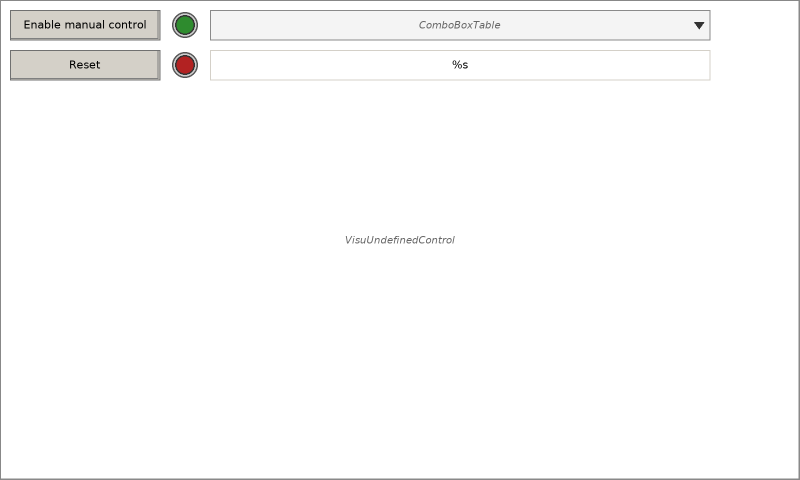
VISUALIZATION ManualControl  // 800x480
VAR_IN_OUT
	stHMI : UDT_HMI_ManualControl;
	fbManualController : FB_ManualController; // Only needed to reference the device array and its size
END_VAR
    Frame (0,0 800x480), input disabled if: NOT stHMI.bEnabled, frame switch variable: stHMI.refSelectedDevice.eDevType
        shows VisuUndefinedControl()
        shows VisuValveControl(pDev := stHMI.pDevValve)
        shows VisuCylinderControl(pDev := stHMI.pDevCylinder)
        shows VisuAxisControl(pDev := stHMI.pDevAxis)
        shows VisuPushbuttonLightControl(pDev := stHMI.pDevPBL)
        shows VisuDigitalInputControl(pDev := stHMI.pDevDigitalInput)
        shows VisuAnlogInputControl(pDev := stHMI.pDevAnalogInput)
        shows VisuDigitalOutControl(pDev := stHMI.pDevDigitalOut)
        shows VisuAnalogOutControl(pDev := stHMI.pDevAnalogOut)
        shows VisuPWMControl(pDev := stHMI.pDevPWMController)
        shows VisuDoublePWMControl(pDev := stHMI.pDevDoublePWM)
        shows VisuEncoderInput(pDev := stHMI.pDevEncoder)
        shows VisuAnalogAxisControl(pDev := stHMI.pDevAnalogAxis)
        shows VisuTwoVelocityAxisControl(pDev := stHMI.pDevTwoVelocityAxis)
        shows VisuKL5151Control(pDev := stHMI.pDevKL5151)
        shows VisuKL15XXControl(pDev := stHMI.pDevKL1512)
        pReferences[2]: HMI=stHMI
        pReferences[3]: HMI=stHMI
        pReferences[4]: HMI=stHMI
        pReferences[5]: HMI=stHMI
        pReferences[6]: HMI=stHMI
        pReferences[7]: HMI=stHMI
        pReferences[8]: HMI=stHMI
        pReferences[9]: HMI=stHMI
        pReferences[10]: HMI=stHMI
        pReferences[11]: HMI=stHMI
        pReferences[12]: HMI=stHMI
        pReferences[13]: HMI=stHMI
        pReferences[14]: HMI=stHMI
        pReferences[15]: HMI=stHMI
    Lamp1 (170,50 30x30), tooltip "component fault active", variable: stHMI.refSelectedDevice.bErrorActive, style: Lamp-Lamp1-Red
    Lamp1 (170,10 30x30), tooltip "Manual control active", variable: stHMI.bEnabled, style: Lamp-Lamp1-Green
    Textfield (210,50 500x30), "%s", text variable: stHMI.refSelectedDevice.sActiveState
    Button (10,50 150x30), "Reset"
        tap stHMI.bReset
    ComboBoxTable (210,10 500x30), variable: stHMI.nSelectedDevice, data array: fbManualController.arDeviceArray
        p1128707560: fbManualController.nNumberOfDevices
        p3854506369: fbManualController.arDeviceArray[INDEX].sName
        p1892666644: fbManualController.arDeviceArray[INDEX].sType
        p338671338: fbManualController.arDeviceArray[INDEX].pFunction^
    Button (10,10 150x30), "Enable manual control"
        toggle stHMI.bEnabled
END_VISUALIZATION

(* stored: Version 1.1.0.1, ProductVersion 3.1.4024.11
   Visu ManualControl: Id {47fd7eab-4722-4161-bb7e-85fd17bf2676} *)
